// TIA Portal V20 export
// export: Created 2025-12-01T14:57:01.7824038Z, ExportSetting None, DisplayName Totally Integrated Automation Portal, DisplayVersion V20 Update 3, DisplayName TIA Portal Openness, DisplayVersion V20 Update 3, DisplayName TIA Portal Version Control Interface, DisplayVersion V20 Update 3, DisplayName STEP 7 Professional, DisplayVersion V20 Update 3, DisplayName STEP 7 Safety, DisplayVersion V20 Update 2, DisplayName WinCC Basic/Comfort/Advanced, DisplayVersion V20 Update 3, DisplayName WinCC Professional, DisplayVersion V20 Update 3, DisplayName WinCC Unified, DisplayVersion V20 Update 3
FUNCTION "FC460_TL_Merge" : Void   // FC460, LAD
{ S7_Optimized_Access := 'FALSE' }
AUTHOR : TLigero
NAME : 20160208
VERSION : 3.3
// stored: AutoNumber false, SetENOAutomatically false
   VAR_INPUT
      Mesa : UInt;
      En_Tension : Bool;
      PhsMx : Bool;
      Avance_Tx : Bool;
      Termico_Tx : Bool;
      Simul_Mx : Bool;
      AVTF_MAnt_E1 : Bool;
      AVTF_MAnt_E2 : Bool;
      PTF_Mx_MSig : Bool;
      NXT_Avance : Bool;
      V_Paro : UDInt;
      V_TOut_Tx_Mx : UDInt;
      V_CNT_pHsMx : UDInt;
      V_Salida : UDInt;
      V_Gap : UDInt;
      V_Cajas_Equ_E1 : UDInt;
      V_Cajas_Equ_E2 : UDInt;
      V_Vaciado_E1 : UDInt;
      V_Vaciado_E2 : UDInt;
   END_VAR
   VAR_OUTPUT
      PTF_Ent_M1 : Bool;
      PTF_Ent_M2 : Bool;
      AVTF_Mx_MSig : Bool;
      NXT_Descarga_Act : Bool;
   END_VAR
   VAR_IN_OUT
      Mem_CNT_Salida : Bool;
      Mem_CNT_Tmp_Paro_Tx : Bool;
      MAUX_FP_Marcha : Bool;
      MAUX_FN_PHS : Bool;
      MAUX_PRV_Carga_OK_E1 : Bool;
      MAUX_PRV_Carga_OK_E2 : Bool;
      MAUX_FP_contador_E1 : Bool;
      MAUX_FP_contador_E2 : Bool;
      MAUX_FP_En_camino_E1 : Bool;
      MAUX_FP_En_camino_E2 : Bool;
      MAUX_key_En_E1 : Bool;
      MAUX_key_En_E2 : Bool;
      MAUX_Key_por_E1_fue_usada : Bool;
      MAUX_Key_por_E2_fue_usada : Bool;
      MAUX_Caja_En_Camino_E1 : Bool;
      MAUX_Caja_En_Camino_E2 : Bool;
   END_VAR
   VAR_TEMP
      OK_Avance : Bool;
      fp_Marcha : Bool;
      fn_phs_tx : Bool;
      fp_phs_tx : Bool;
      Mem_CNT_Centrado : Bool;
      Mem_CNT_Gap : Bool;
      Error_atasco : Bool;
      TEMP_NXT_AVTF : Bool;
      TEMP_PRV_CARGA_OK : Bool;
      VaciadoE1_OK : Bool;
      VaciadoE2_OK : Bool;
      ok_tension : Bool;
   END_VAR
   VAR_TEMP   // added for the SCL form of the ladder/FBD networks
      _w1 : Bool;
   END_VAR
BEGIN

REGION Network 1: Marca General Error
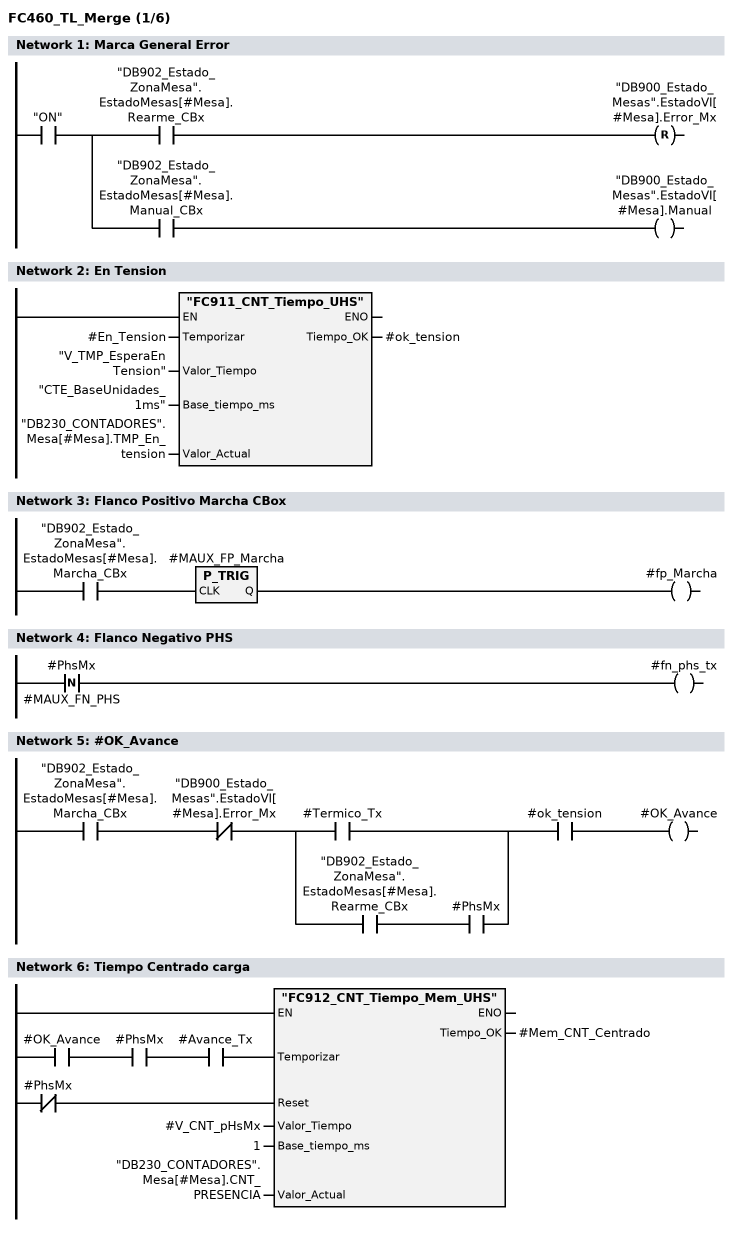
   RUNG wire#powerrail
      Contact( "ON" )
      wire#w1
      Contact( "DB902_Estado_ZonaMesa".EstadoMesas[#Mesa].Rearme_CBx )
      R_Coil( "DB900_Estado_Mesas".EstadoVI[#Mesa].Error_Mx )
   END_RUNG
   RUNG wire#w1
      Contact( "DB902_Estado_ZonaMesa".EstadoMesas[#Mesa].Manual_CBx )
      Coil( "DB900_Estado_Mesas".EstadoVI[#Mesa].Manual )
   END_RUNG
   // the same network as SCL:
   IF "ON" AND "DB902_Estado_ZonaMesa".EstadoMesas[#Mesa].Rearme_CBx THEN
       "DB900_Estado_Mesas".EstadoVI[#Mesa].Error_Mx := FALSE;
   END_IF;
   "DB900_Estado_Mesas".EstadoVI[#Mesa].Manual := "ON" AND "DB902_Estado_ZonaMesa".EstadoMesas[#Mesa].Manual_CBx;
END_REGION

REGION Network 2: En Tension
   RUNG wire#powerrail
      "FC911_CNT_Tiempo_UHS"(Temporizar := #En_Tension, Valor_Tiempo := "V_TMP_EsperaEnTension", Base_tiempo_ms := "CTE_BaseUnidades_1ms", Valor_Actual := "DB230_CONTADORES".Mesa[#Mesa].TMP_En_tension, Tiempo_OK => #ok_tension)
   END_RUNG
   // the same network as SCL:
   "FC911_CNT_Tiempo_UHS"(Temporizar := #En_Tension,
                          Valor_Tiempo := "V_TMP_EsperaEnTension",
                          Base_tiempo_ms := "CTE_BaseUnidades_1ms",
                          Valor_Actual := "DB230_CONTADORES".Mesa[#Mesa].TMP_En_tension,
                          Tiempo_OK => #ok_tension);
END_REGION

REGION Network 3: Flanco Positivo Marcha CBox
   RUNG wire#powerrail
      Contact( "DB902_Estado_ZonaMesa".EstadoMesas[#Mesa].Marcha_CBx )
      P_Trig( #MAUX_FP_Marcha )
      Coil( #fp_Marcha )
   END_RUNG
   // the same network as SCL:
   #_w1 := "DB902_Estado_ZonaMesa".EstadoMesas[#Mesa].Marcha_CBx AND NOT #MAUX_FP_Marcha;   // rising edge
   #MAUX_FP_Marcha := "DB902_Estado_ZonaMesa".EstadoMesas[#Mesa].Marcha_CBx;
   #fp_Marcha := #_w1;
END_REGION

REGION Network 4: Flanco Negativo PHS
   RUNG wire#powerrail
      N_Contact(operand := #PhsMx, bit := #MAUX_FN_PHS)
      Coil( #fn_phs_tx )
   END_RUNG
   // the same network as SCL:
   #_w1 := NOT #PhsMx AND #MAUX_FN_PHS;   // falling edge of #PhsMx
   #MAUX_FN_PHS := #PhsMx;
   #fn_phs_tx := #_w1;
END_REGION

REGION Network 5: #OK_Avance
   RUNG wire#powerrail
      Contact( "DB902_Estado_ZonaMesa".EstadoMesas[#Mesa].Marcha_CBx )
      I_Contact( "DB900_Estado_Mesas".EstadoVI[#Mesa].Error_Mx )
      wire#w1
      Contact( #Termico_Tx )
      wire#w2
      Contact( #ok_tension )
      Coil( #OK_Avance )
   END_RUNG
   RUNG wire#w1
      Contact( "DB902_Estado_ZonaMesa".EstadoMesas[#Mesa].Rearme_CBx )
      Contact( #PhsMx )
   END_RUNG wire#w2
   // the same network as SCL:
   #OK_Avance := "DB902_Estado_ZonaMesa".EstadoMesas[#Mesa].Marcha_CBx AND NOT "DB900_Estado_Mesas".EstadoVI[#Mesa].Error_Mx AND (#Termico_Tx OR ("DB902_Estado_ZonaMesa".EstadoMesas[#Mesa].Rearme_CBx AND #PhsMx)) AND #ok_tension;
END_REGION

REGION Network 6: Tiempo Centrado carga
   RUNG wire#powerrail
      "FC912_CNT_Tiempo_Mem_UHS"(Temporizar := wire#w1, Reset := wire#w2, Valor_Tiempo := #V_CNT_pHsMx, Base_tiempo_ms := 1, Valor_Actual := "DB230_CONTADORES".Mesa[#Mesa].CNT_PRESENCIA, Tiempo_OK => #Mem_CNT_Centrado)
   END_RUNG
   RUNG wire#powerrail
      Contact( #OK_Avance )
      Contact( #PhsMx )
      Contact( #Avance_Tx )
   END_RUNG wire#w1
   RUNG wire#powerrail
      I_Contact( #PhsMx )
   END_RUNG wire#w2
   // the same network as SCL:
   "FC912_CNT_Tiempo_Mem_UHS"(Temporizar := #OK_Avance AND #PhsMx AND #Avance_Tx,
                           Reset := NOT #PhsMx,
                           Valor_Tiempo := #V_CNT_pHsMx,
                           Base_tiempo_ms := 1,
                           Valor_Actual := "DB230_CONTADORES".Mesa[#Mesa].CNT_PRESENCIA,
                           Tiempo_OK => #Mem_CNT_Centrado);
END_REGION

REGION Network 7: Tiempo Centrado carga
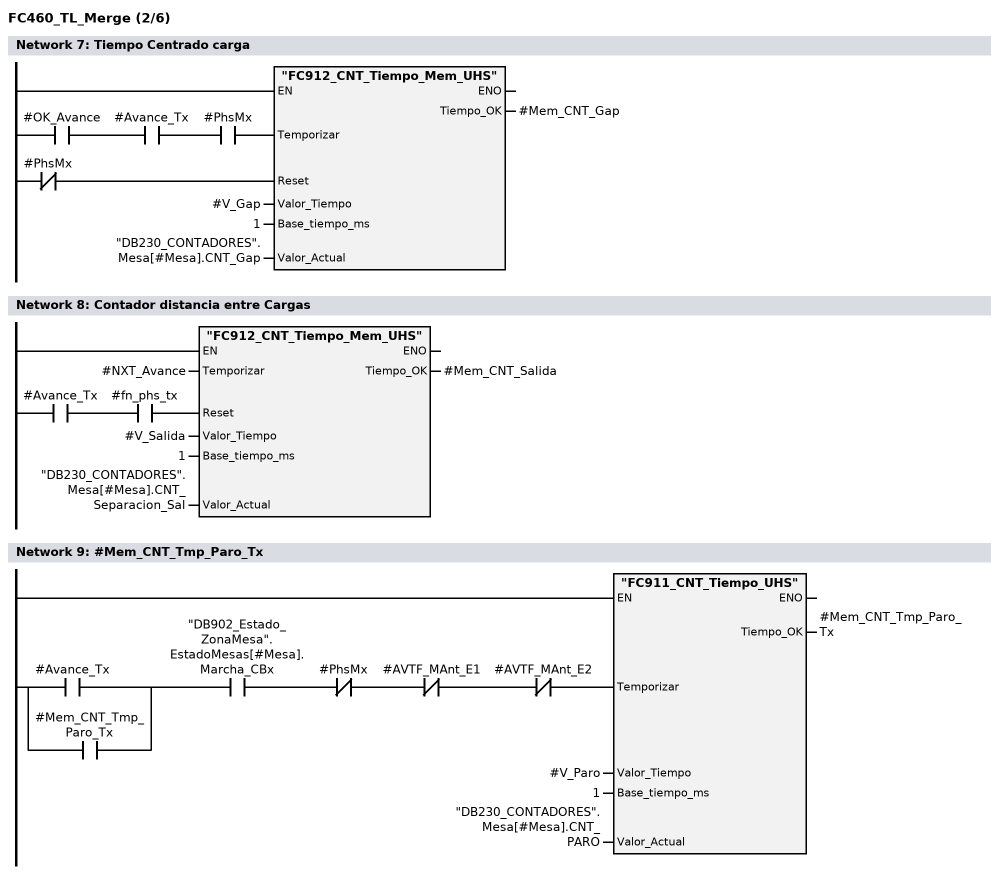
   RUNG wire#powerrail
      "FC912_CNT_Tiempo_Mem_UHS"(Temporizar := wire#w1, Reset := wire#w2, Valor_Tiempo := #V_Gap, Base_tiempo_ms := 1, Valor_Actual := "DB230_CONTADORES".Mesa[#Mesa].CNT_Gap, Tiempo_OK => #Mem_CNT_Gap)
   END_RUNG
   RUNG wire#powerrail
      Contact( #OK_Avance )
      Contact( #Avance_Tx )
      Contact( #PhsMx )
   END_RUNG wire#w1
   RUNG wire#powerrail
      I_Contact( #PhsMx )
   END_RUNG wire#w2
   // the same network as SCL:
   "FC912_CNT_Tiempo_Mem_UHS"(Temporizar := #OK_Avance AND #Avance_Tx AND #PhsMx,
                           Reset := NOT #PhsMx,
                           Valor_Tiempo := #V_Gap,
                           Base_tiempo_ms := 1,
                           Valor_Actual := "DB230_CONTADORES".Mesa[#Mesa].CNT_Gap,
                           Tiempo_OK => #Mem_CNT_Gap);
END_REGION

REGION Network 8: Contador distancia entre Cargas
   RUNG wire#powerrail
      "FC912_CNT_Tiempo_Mem_UHS"(Reset := wire#w1, Temporizar := #NXT_Avance, Valor_Tiempo := #V_Salida, Base_tiempo_ms := 1, Valor_Actual := "DB230_CONTADORES".Mesa[#Mesa].CNT_Separacion_Sal, Tiempo_OK => #Mem_CNT_Salida)
   END_RUNG
   RUNG wire#powerrail
      Contact( #Avance_Tx )
      Contact( #fn_phs_tx )
   END_RUNG wire#w1
   // the same network as SCL:
   "FC912_CNT_Tiempo_Mem_UHS"(Temporizar := #NXT_Avance,
                           Reset := #Avance_Tx AND #fn_phs_tx,
                           Valor_Tiempo := #V_Salida,
                           Base_tiempo_ms := 1,
                           Valor_Actual := "DB230_CONTADORES".Mesa[#Mesa].CNT_Separacion_Sal,
                           Tiempo_OK => #Mem_CNT_Salida);
END_REGION

REGION Network 9: #Mem_CNT_Tmp_Paro_Tx
   RUNG wire#powerrail
      "FC911_CNT_Tiempo_UHS"(Temporizar := wire#w2, Valor_Tiempo := #V_Paro, Base_tiempo_ms := 1, Valor_Actual := "DB230_CONTADORES".Mesa[#Mesa].CNT_PARO, Tiempo_OK => #Mem_CNT_Tmp_Paro_Tx)
   END_RUNG
   RUNG wire#powerrail
      Contact( #Avance_Tx )
      wire#w1
      Contact( "DB902_Estado_ZonaMesa".EstadoMesas[#Mesa].Marcha_CBx )
      I_Contact( #PhsMx )
      I_Contact( #AVTF_MAnt_E1 )
      I_Contact( #AVTF_MAnt_E2 )
   END_RUNG wire#w2
   RUNG wire#powerrail
      Contact( #Mem_CNT_Tmp_Paro_Tx )
   END_RUNG wire#w1
   // the same network as SCL:
   "FC911_CNT_Tiempo_UHS"(Temporizar := (#Avance_Tx OR #Mem_CNT_Tmp_Paro_Tx) AND "DB902_Estado_ZonaMesa".EstadoMesas[#Mesa].Marcha_CBx AND NOT #PhsMx AND NOT #AVTF_MAnt_E1 AND NOT #AVTF_MAnt_E2,
                          Valor_Tiempo := #V_Paro,
                          Base_tiempo_ms := 1,
                          Valor_Actual := "DB230_CONTADORES".Mesa[#Mesa].CNT_PARO,
                          Tiempo_OK => #Mem_CNT_Tmp_Paro_Tx);
END_REGION

REGION Network 10: #MA_AV_13_T_MX
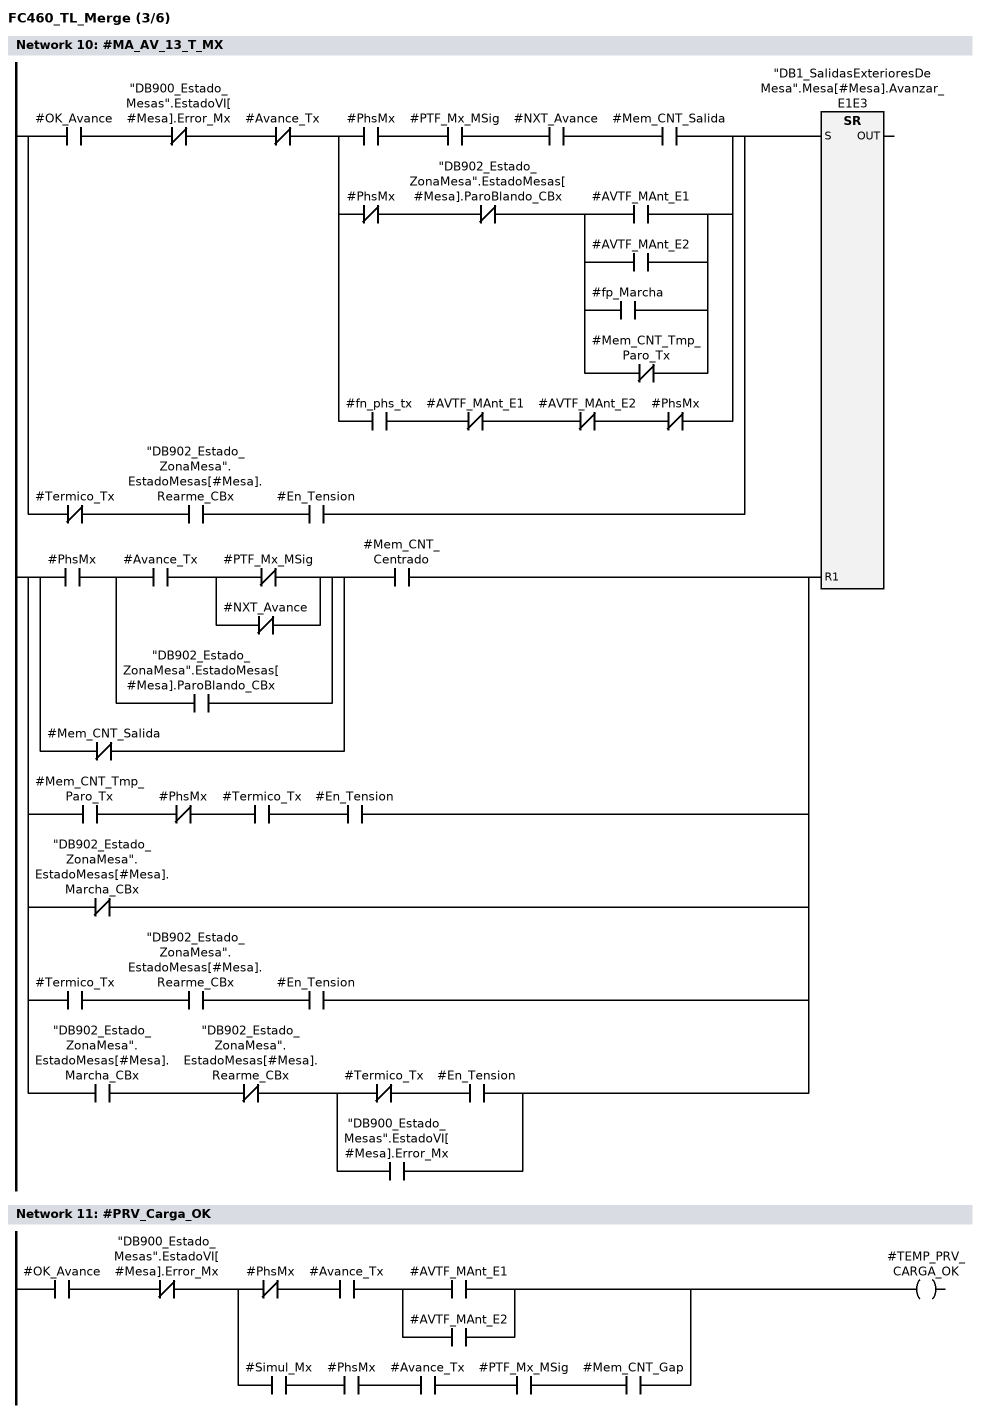
   RUNG wire#powerrail
      Contact( #OK_Avance )
      I_Contact( "DB900_Estado_Mesas".EstadoVI[#Mesa].Error_Mx )
      I_Contact( #Avance_Tx )
      wire#w1
      Contact( #PhsMx )
      Contact( #PTF_Mx_MSig )
      Contact( #NXT_Avance )
      Contact( #Mem_CNT_Salida )
      wire#w2
      S_SR(operand := "DB1_SalidasExterioresDeMesa".Mesa[#Mesa].Avanzar_E1E3, r1 := wire#w8)
   END_RUNG
   RUNG wire#w1
      I_Contact( #PhsMx )
      I_Contact( "DB902_Estado_ZonaMesa".EstadoMesas[#Mesa].ParoBlando_CBx )
      wire#w3
      Contact( #AVTF_MAnt_E1 )
   END_RUNG wire#w2
   RUNG wire#w3
      Contact( #AVTF_MAnt_E2 )
   END_RUNG wire#w2
   RUNG wire#w3
      Contact( #fp_Marcha )
   END_RUNG wire#w2
   RUNG wire#w3
      I_Contact( #Mem_CNT_Tmp_Paro_Tx )
   END_RUNG wire#w2
   RUNG wire#w1
      Contact( #fn_phs_tx )
      I_Contact( #AVTF_MAnt_E1 )
      I_Contact( #AVTF_MAnt_E2 )
      I_Contact( #PhsMx )
   END_RUNG wire#w2
   RUNG wire#powerrail
      I_Contact( #Termico_Tx )
      Contact( "DB902_Estado_ZonaMesa".EstadoMesas[#Mesa].Rearme_CBx )
      Contact( #En_Tension )
   END_RUNG wire#w2
   RUNG wire#powerrail
      Contact( #PhsMx )
      wire#w4
      Contact( #Avance_Tx )
      wire#w5
      I_Contact( #PTF_Mx_MSig )
      wire#w6
      Contact( #Mem_CNT_Centrado )
   END_RUNG wire#w8
   RUNG wire#w5
      I_Contact( #NXT_Avance )
   END_RUNG wire#w6
   RUNG wire#w4
      Contact( "DB902_Estado_ZonaMesa".EstadoMesas[#Mesa].ParoBlando_CBx )
   END_RUNG wire#w6
   RUNG wire#powerrail
      I_Contact( #Mem_CNT_Salida )
   END_RUNG wire#w6
   RUNG wire#powerrail
      Contact( #Mem_CNT_Tmp_Paro_Tx )
      I_Contact( #PhsMx )
      Contact( #Termico_Tx )
      Contact( #En_Tension )
   END_RUNG wire#w8
   RUNG wire#powerrail
      I_Contact( "DB902_Estado_ZonaMesa".EstadoMesas[#Mesa].Marcha_CBx )
   END_RUNG wire#w8
   RUNG wire#powerrail
      Contact( #Termico_Tx )
      Contact( "DB902_Estado_ZonaMesa".EstadoMesas[#Mesa].Rearme_CBx )
      Contact( #En_Tension )
   END_RUNG wire#w8
   RUNG wire#powerrail
      Contact( "DB902_Estado_ZonaMesa".EstadoMesas[#Mesa].Marcha_CBx )
      I_Contact( "DB902_Estado_ZonaMesa".EstadoMesas[#Mesa].Rearme_CBx )
      wire#w7
      I_Contact( #Termico_Tx )
      Contact( #En_Tension )
   END_RUNG wire#w8
   RUNG wire#w7
      Contact( "DB900_Estado_Mesas".EstadoVI[#Mesa].Error_Mx )
   END_RUNG wire#w8
   // the same network as SCL:
   #_w1 := (((#PhsMx AND ((#Avance_Tx AND (NOT #PTF_Mx_MSig OR NOT #NXT_Avance)) OR "DB902_Estado_ZonaMesa".EstadoMesas[#Mesa].ParoBlando_CBx)) OR NOT #Mem_CNT_Salida) AND #Mem_CNT_Centrado) OR (#Mem_CNT_Tmp_Paro_Tx AND NOT #PhsMx AND #Termico_Tx AND #En_Tension) OR NOT "DB902_Estado_ZonaMesa".EstadoMesas[#Mesa].Marcha_CBx OR (#Termico_Tx AND "DB902_Estado_ZonaMesa".EstadoMesas[#Mesa].Rearme_CBx AND #En_Tension) OR ("DB902_Estado_ZonaMesa".EstadoMesas[#Mesa].Marcha_CBx AND NOT "DB902_Estado_ZonaMesa".EstadoMesas[#Mesa].Rearme_CBx AND ((NOT #Termico_Tx AND #En_Tension) OR "DB900_Estado_Mesas".EstadoVI[#Mesa].Error_Mx));
   IF (#OK_Avance AND NOT "DB900_Estado_Mesas".EstadoVI[#Mesa].Error_Mx AND NOT #Avance_Tx AND ((#PhsMx AND #PTF_Mx_MSig AND #NXT_Avance AND #Mem_CNT_Salida) OR (NOT #PhsMx AND NOT "DB902_Estado_ZonaMesa".EstadoMesas[#Mesa].ParoBlando_CBx AND (#AVTF_MAnt_E1 OR #AVTF_MAnt_E2 OR #fp_Marcha OR NOT #Mem_CNT_Tmp_Paro_Tx)) OR (#fn_phs_tx AND NOT #AVTF_MAnt_E1 AND NOT #AVTF_MAnt_E2 AND NOT #PhsMx))) OR (NOT #Termico_Tx AND "DB902_Estado_ZonaMesa".EstadoMesas[#Mesa].Rearme_CBx AND #En_Tension) THEN
       "DB1_SalidasExterioresDeMesa".Mesa[#Mesa].Avanzar_E1E3 := TRUE;   // SR flip-flop
   END_IF;
   IF #_w1 THEN "DB1_SalidasExterioresDeMesa".Mesa[#Mesa].Avanzar_E1E3 := FALSE; END_IF;
END_REGION

REGION Network 11: #PRV_Carga_OK
   RUNG wire#powerrail
      Contact( #OK_Avance )
      I_Contact( "DB900_Estado_Mesas".EstadoVI[#Mesa].Error_Mx )
      wire#w1
      I_Contact( #PhsMx )
      Contact( #Avance_Tx )
      wire#w2
      Contact( #AVTF_MAnt_E1 )
      wire#w3
      Coil( #TEMP_PRV_CARGA_OK )
   END_RUNG
   RUNG wire#w2
      Contact( #AVTF_MAnt_E2 )
   END_RUNG wire#w3
   RUNG wire#w1
      Contact( #Simul_Mx )
      Contact( #PhsMx )
      Contact( #Avance_Tx )
      Contact( #PTF_Mx_MSig )
      Contact( #Mem_CNT_Gap )
   END_RUNG wire#w3
   // the same network as SCL:
   #TEMP_PRV_CARGA_OK := #OK_Avance AND NOT "DB900_Estado_Mesas".EstadoVI[#Mesa].Error_Mx AND ((NOT #PhsMx AND #Avance_Tx AND (#AVTF_MAnt_E1 OR #AVTF_MAnt_E2)) OR (#Simul_Mx AND #PhsMx AND #Avance_Tx AND #PTF_Mx_MSig AND #Mem_CNT_Gap));
END_REGION

REGION Network 12: #NXT_AVTF
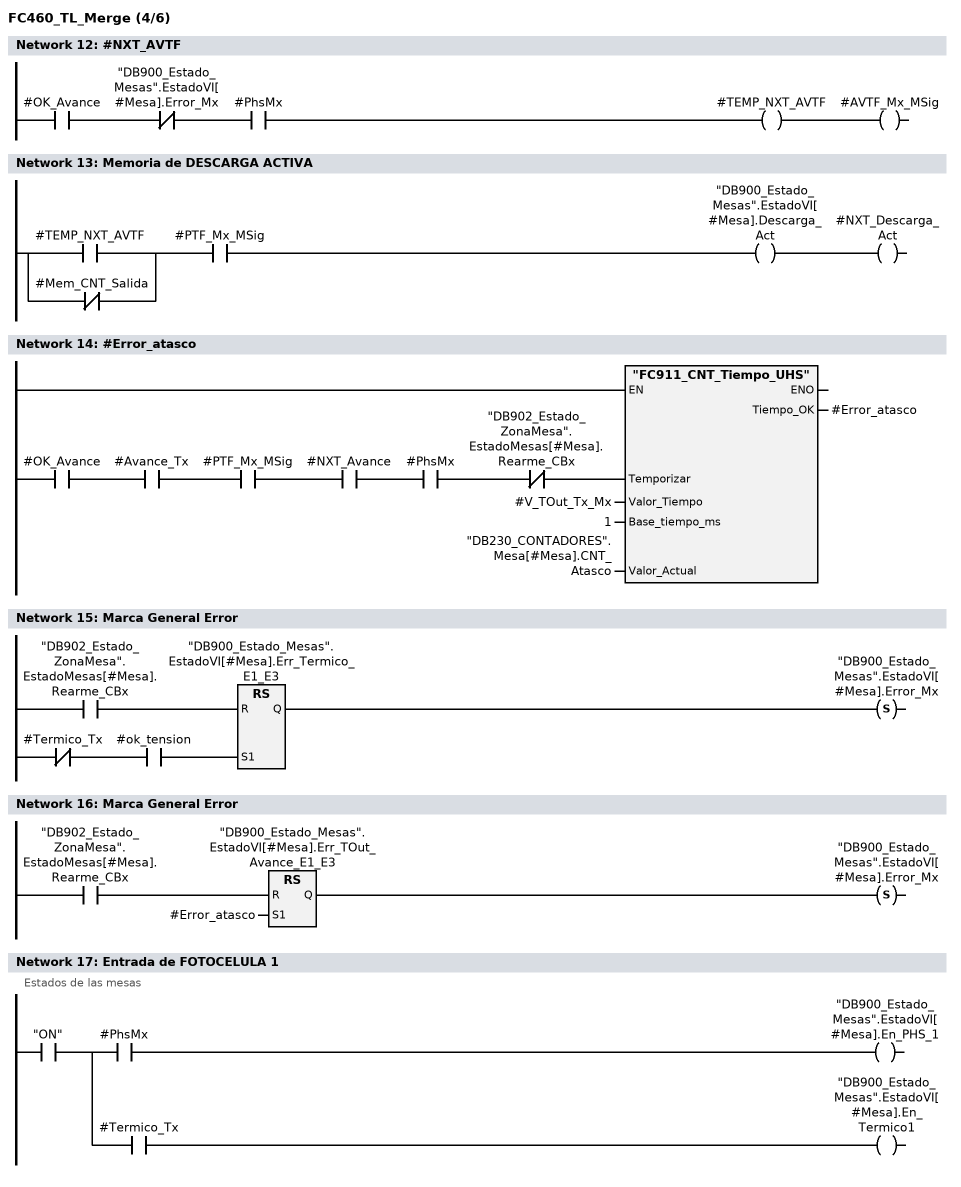
   RUNG wire#powerrail
      Contact( #OK_Avance )
      I_Contact( "DB900_Estado_Mesas".EstadoVI[#Mesa].Error_Mx )
      Contact( #PhsMx )
      Coil( #TEMP_NXT_AVTF )
      Coil( #AVTF_Mx_MSig )
   END_RUNG
   // the same network as SCL:
   #TEMP_NXT_AVTF := #OK_Avance AND NOT "DB900_Estado_Mesas".EstadoVI[#Mesa].Error_Mx AND #PhsMx;
   #AVTF_Mx_MSig := #TEMP_NXT_AVTF;
END_REGION

REGION Network 13: Memoria de DESCARGA ACTIVA
   RUNG wire#powerrail
      Contact( #TEMP_NXT_AVTF )
      wire#w1
      Contact( #PTF_Mx_MSig )
      Coil( "DB900_Estado_Mesas".EstadoVI[#Mesa].Descarga_Act )
      Coil( #NXT_Descarga_Act )
   END_RUNG
   RUNG wire#powerrail
      I_Contact( #Mem_CNT_Salida )
   END_RUNG wire#w1
   // the same network as SCL:
   "DB900_Estado_Mesas".EstadoVI[#Mesa].Descarga_Act := (#TEMP_NXT_AVTF OR NOT #Mem_CNT_Salida) AND #PTF_Mx_MSig;
   #NXT_Descarga_Act := (#TEMP_NXT_AVTF OR NOT #Mem_CNT_Salida) AND #PTF_Mx_MSig;
END_REGION

REGION Network 14: #Error_atasco
   RUNG wire#powerrail
      "FC911_CNT_Tiempo_UHS"(Temporizar := wire#w1, Valor_Tiempo := #V_TOut_Tx_Mx, Base_tiempo_ms := 1, Valor_Actual := "DB230_CONTADORES".Mesa[#Mesa].CNT_Atasco, Tiempo_OK => #Error_atasco)
   END_RUNG
   RUNG wire#powerrail
      Contact( #OK_Avance )
      Contact( #Avance_Tx )
      Contact( #PTF_Mx_MSig )
      Contact( #NXT_Avance )
      Contact( #PhsMx )
      I_Contact( "DB902_Estado_ZonaMesa".EstadoMesas[#Mesa].Rearme_CBx )
   END_RUNG wire#w1
   // the same network as SCL:
   "FC911_CNT_Tiempo_UHS"(Temporizar := #OK_Avance AND #Avance_Tx AND #PTF_Mx_MSig AND #NXT_Avance AND #PhsMx AND NOT "DB902_Estado_ZonaMesa".EstadoMesas[#Mesa].Rearme_CBx,
                          Valor_Tiempo := #V_TOut_Tx_Mx,
                          Base_tiempo_ms := 1,
                          Valor_Actual := "DB230_CONTADORES".Mesa[#Mesa].CNT_Atasco,
                          Tiempo_OK => #Error_atasco);
END_REGION

REGION Network 15: Marca General Error
   RUNG wire#powerrail
      Contact( "DB902_Estado_ZonaMesa".EstadoMesas[#Mesa].Rearme_CBx )
      S_RS(operand := "DB900_Estado_Mesas".EstadoVI[#Mesa].Err_Termico_E1_E3, s1 := wire#w1)
      S_Coil( "DB900_Estado_Mesas".EstadoVI[#Mesa].Error_Mx )
   END_RUNG
   RUNG wire#powerrail
      I_Contact( #Termico_Tx )
      Contact( #ok_tension )
   END_RUNG wire#w1
   // the same network as SCL:
   IF "DB902_Estado_ZonaMesa".EstadoMesas[#Mesa].Rearme_CBx THEN
       "DB900_Estado_Mesas".EstadoVI[#Mesa].Err_Termico_E1_E3 := FALSE;   // RS flip-flop
   END_IF;
   IF NOT #Termico_Tx AND #ok_tension THEN
       "DB900_Estado_Mesas".EstadoVI[#Mesa].Err_Termico_E1_E3 := TRUE;
   END_IF;
   IF "DB900_Estado_Mesas".EstadoVI[#Mesa].Err_Termico_E1_E3 THEN
       "DB900_Estado_Mesas".EstadoVI[#Mesa].Error_Mx := TRUE;
   END_IF;
END_REGION

REGION Network 16: Marca General Error
   RUNG wire#powerrail
      Contact( "DB902_Estado_ZonaMesa".EstadoMesas[#Mesa].Rearme_CBx )
      S_RS(operand := "DB900_Estado_Mesas".EstadoVI[#Mesa].Err_TOut_Avance_E1_E3, s1 := #Error_atasco)
      S_Coil( "DB900_Estado_Mesas".EstadoVI[#Mesa].Error_Mx )
   END_RUNG
   // the same network as SCL:
   IF "DB902_Estado_ZonaMesa".EstadoMesas[#Mesa].Rearme_CBx THEN
       "DB900_Estado_Mesas".EstadoVI[#Mesa].Err_TOut_Avance_E1_E3 := FALSE;   // RS flip-flop
   END_IF;
   IF #Error_atasco THEN "DB900_Estado_Mesas".EstadoVI[#Mesa].Err_TOut_Avance_E1_E3 := TRUE; END_IF;
   IF "DB900_Estado_Mesas".EstadoVI[#Mesa].Err_TOut_Avance_E1_E3 THEN
       "DB900_Estado_Mesas".EstadoVI[#Mesa].Error_Mx := TRUE;
   END_IF;
END_REGION

REGION Network 17: Entrada de FOTOCELULA 1
   // Estados de las mesas
   RUNG wire#powerrail
      Contact( "ON" )
      wire#w1
      Contact( #PhsMx )
      Coil( "DB900_Estado_Mesas".EstadoVI[#Mesa].En_PHS_1 )
   END_RUNG
   RUNG wire#w1
      Contact( #Termico_Tx )
      Coil( "DB900_Estado_Mesas".EstadoVI[#Mesa].En_Termico1 )
   END_RUNG
   // the same network as SCL:
   "DB900_Estado_Mesas".EstadoVI[#Mesa].En_PHS_1 := "ON" AND #PhsMx;
   "DB900_Estado_Mesas".EstadoVI[#Mesa].En_Termico1 := "ON" AND #Termico_Tx;
END_REGION

REGION Network 18: ESTADOS MESA 1
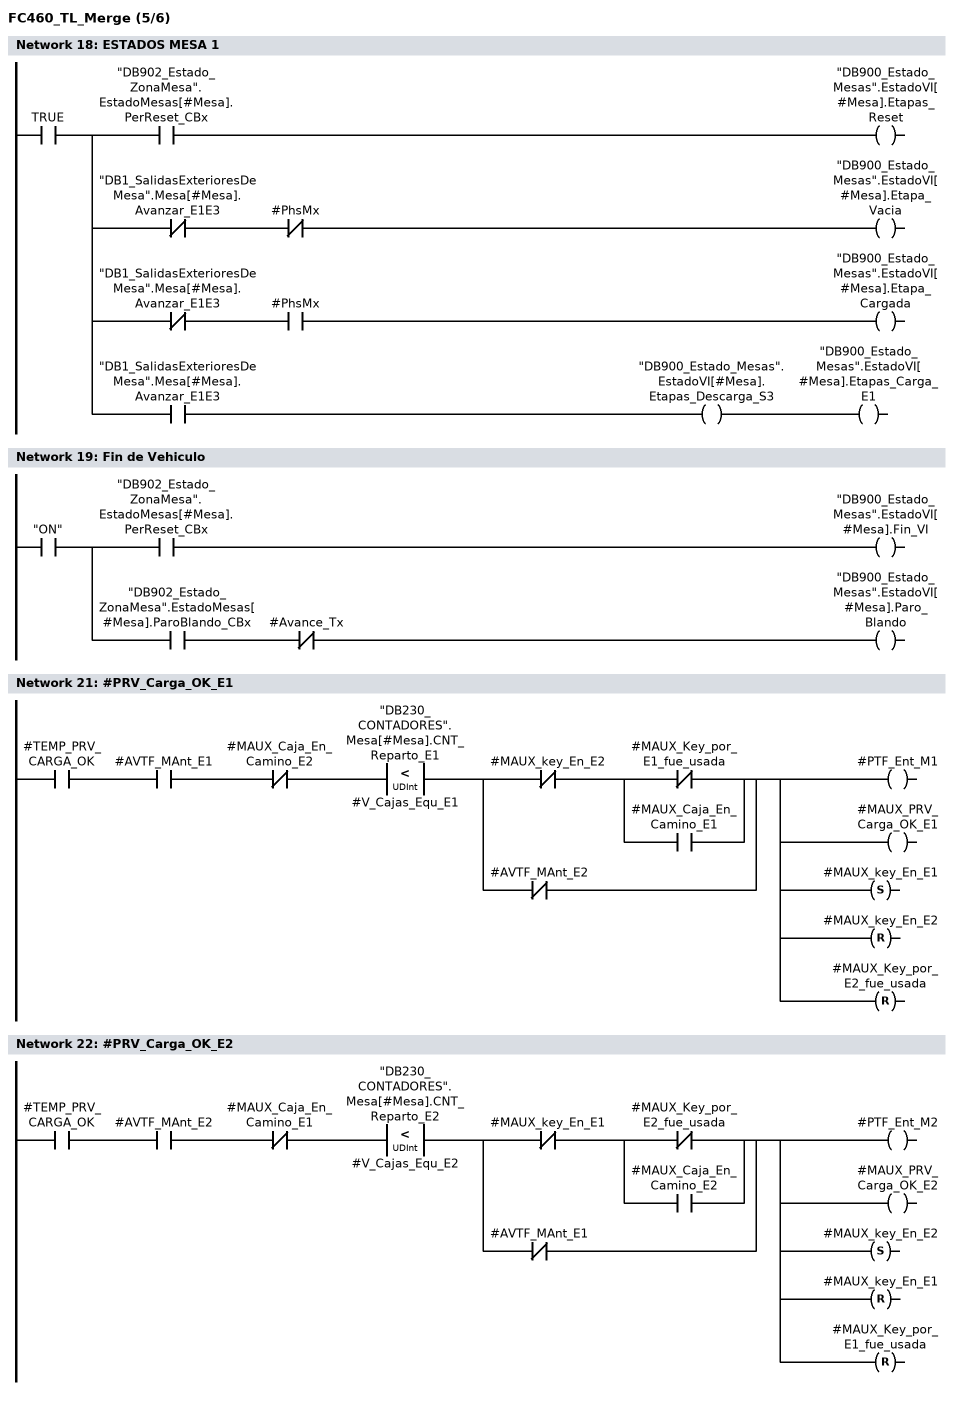
   RUNG wire#powerrail
      Contact( TRUE )
      wire#w1
      Contact( "DB902_Estado_ZonaMesa".EstadoMesas[#Mesa].PerReset_CBx )
      Coil( "DB900_Estado_Mesas".EstadoVI[#Mesa].Etapas_Reset )
   END_RUNG
   RUNG wire#w1
      I_Contact( "DB1_SalidasExterioresDeMesa".Mesa[#Mesa].Avanzar_E1E3 )
      I_Contact( #PhsMx )
      Coil( "DB900_Estado_Mesas".EstadoVI[#Mesa].Etapa_Vacia )
   END_RUNG
   RUNG wire#w1
      I_Contact( "DB1_SalidasExterioresDeMesa".Mesa[#Mesa].Avanzar_E1E3 )
      Contact( #PhsMx )
      Coil( "DB900_Estado_Mesas".EstadoVI[#Mesa].Etapa_Cargada )
   END_RUNG
   RUNG wire#w1
      Contact( "DB1_SalidasExterioresDeMesa".Mesa[#Mesa].Avanzar_E1E3 )
      Coil( "DB900_Estado_Mesas".EstadoVI[#Mesa].Etapas_Descarga_S3 )
      Coil( "DB900_Estado_Mesas".EstadoVI[#Mesa].Etapas_Carga_E1 )
   END_RUNG
   // the same network as SCL:
   "DB900_Estado_Mesas".EstadoVI[#Mesa].Etapas_Reset := TRUE AND "DB902_Estado_ZonaMesa".EstadoMesas[#Mesa].PerReset_CBx;
   "DB900_Estado_Mesas".EstadoVI[#Mesa].Etapa_Vacia := TRUE AND NOT "DB1_SalidasExterioresDeMesa".Mesa[#Mesa].Avanzar_E1E3 AND NOT #PhsMx;
   "DB900_Estado_Mesas".EstadoVI[#Mesa].Etapa_Cargada := TRUE AND NOT "DB1_SalidasExterioresDeMesa".Mesa[#Mesa].Avanzar_E1E3 AND #PhsMx;
   #_w1 := TRUE AND "DB1_SalidasExterioresDeMesa".Mesa[#Mesa].Avanzar_E1E3;
   "DB900_Estado_Mesas".EstadoVI[#Mesa].Etapas_Descarga_S3 := #_w1;
   "DB900_Estado_Mesas".EstadoVI[#Mesa].Etapas_Carga_E1 := #_w1;
END_REGION

REGION Network 19: Fin de Vehiculo
   RUNG wire#powerrail
      Contact( "ON" )
      wire#w1
      Contact( "DB902_Estado_ZonaMesa".EstadoMesas[#Mesa].PerReset_CBx )
      Coil( "DB900_Estado_Mesas".EstadoVI[#Mesa].Fin_VI )
   END_RUNG
   RUNG wire#w1
      Contact( "DB902_Estado_ZonaMesa".EstadoMesas[#Mesa].ParoBlando_CBx )
      I_Contact( #Avance_Tx )
      Coil( "DB900_Estado_Mesas".EstadoVI[#Mesa].Paro_Blando )
   END_RUNG
   // the same network as SCL:
   "DB900_Estado_Mesas".EstadoVI[#Mesa].Fin_VI := "ON" AND "DB902_Estado_ZonaMesa".EstadoMesas[#Mesa].PerReset_CBx;
   "DB900_Estado_Mesas".EstadoVI[#Mesa].Paro_Blando := "ON" AND "DB902_Estado_ZonaMesa".EstadoMesas[#Mesa].ParoBlando_CBx AND NOT #Avance_Tx;
END_REGION

REGION Network 20: Gestion de cruce
END_REGION

REGION Network 21: #PRV_Carga_OK_E1
   RUNG wire#powerrail
      Contact( #TEMP_PRV_CARGA_OK )
      Contact( #AVTF_MAnt_E1 )
      I_Contact( #MAUX_Caja_En_Camino_E2 )
      { S7_Templates := "SrcType := UDInt" } LT_Contact(in1 := "DB230_CONTADORES".Mesa[#Mesa].CNT_Reparto_E1, in2 := #V_Cajas_Equ_E1)
      wire#w1
      I_Contact( #MAUX_key_En_E2 )
      wire#w2
      I_Contact( #MAUX_Key_por_E1_fue_usada )
      wire#w3
      Coil( #PTF_Ent_M1 )
   END_RUNG
   RUNG wire#w2
      Contact( #MAUX_Caja_En_Camino_E1 )
   END_RUNG wire#w3
   RUNG wire#w1
      I_Contact( #AVTF_MAnt_E2 )
   END_RUNG wire#w3
   RUNG wire#w3
      Coil( #MAUX_PRV_Carga_OK_E1 )
   END_RUNG
   RUNG wire#w3
      S_Coil( #MAUX_key_En_E1 )
   END_RUNG
   RUNG wire#w3
      R_Coil( #MAUX_key_En_E2 )
   END_RUNG
   RUNG wire#w3
      R_Coil( #MAUX_Key_por_E2_fue_usada )
   END_RUNG
   // the same network as SCL:
   #PTF_Ent_M1 := #TEMP_PRV_CARGA_OK AND #AVTF_MAnt_E1 AND NOT #MAUX_Caja_En_Camino_E2 AND ("DB230_CONTADORES".Mesa[#Mesa].CNT_Reparto_E1 < #V_Cajas_Equ_E1) AND ((NOT #MAUX_key_En_E2 AND (NOT #MAUX_Key_por_E1_fue_usada OR #MAUX_Caja_En_Camino_E1)) OR NOT #AVTF_MAnt_E2);
   #MAUX_PRV_Carga_OK_E1 := #PTF_Ent_M1;
   IF #PTF_Ent_M1 THEN
       #MAUX_key_En_E1 := TRUE;
       #MAUX_key_En_E2 := FALSE;
       #MAUX_Key_por_E2_fue_usada := FALSE;
   END_IF;
END_REGION

REGION Network 22: #PRV_Carga_OK_E2
   RUNG wire#powerrail
      Contact( #TEMP_PRV_CARGA_OK )
      Contact( #AVTF_MAnt_E2 )
      I_Contact( #MAUX_Caja_En_Camino_E1 )
      { S7_Templates := "SrcType := UDInt" } LT_Contact(in1 := "DB230_CONTADORES".Mesa[#Mesa].CNT_Reparto_E2, in2 := #V_Cajas_Equ_E2)
      wire#w1
      I_Contact( #MAUX_key_En_E1 )
      wire#w2
      I_Contact( #MAUX_Key_por_E2_fue_usada )
      wire#w3
      Coil( #PTF_Ent_M2 )
   END_RUNG
   RUNG wire#w2
      Contact( #MAUX_Caja_En_Camino_E2 )
   END_RUNG wire#w3
   RUNG wire#w1
      I_Contact( #AVTF_MAnt_E1 )
   END_RUNG wire#w3
   RUNG wire#w3
      Coil( #MAUX_PRV_Carga_OK_E2 )
   END_RUNG
   RUNG wire#w3
      S_Coil( #MAUX_key_En_E2 )
   END_RUNG
   RUNG wire#w3
      R_Coil( #MAUX_key_En_E1 )
   END_RUNG
   RUNG wire#w3
      R_Coil( #MAUX_Key_por_E1_fue_usada )
   END_RUNG
   // the same network as SCL:
   #PTF_Ent_M2 := #TEMP_PRV_CARGA_OK AND #AVTF_MAnt_E2 AND NOT #MAUX_Caja_En_Camino_E1 AND ("DB230_CONTADORES".Mesa[#Mesa].CNT_Reparto_E2 < #V_Cajas_Equ_E2) AND ((NOT #MAUX_key_En_E1 AND (NOT #MAUX_Key_por_E2_fue_usada OR #MAUX_Caja_En_Camino_E2)) OR NOT #AVTF_MAnt_E1);
   #MAUX_PRV_Carga_OK_E2 := #PTF_Ent_M2;
   IF #PTF_Ent_M2 THEN
       #MAUX_key_En_E2 := TRUE;
       #MAUX_key_En_E1 := FALSE;
       #MAUX_Key_por_E1_fue_usada := FALSE;
   END_IF;
END_REGION

NETWORK
TITLE = Contador de cajas permitidas por E1
      A     #MAUX_PRV_Carga_OK_E1;
      FN    #MAUX_FP_contador_E1;
      JCN   cont1;

      L     "DB230_CONTADORES".Mesa[#Mesa].CNT_Reparto_E1;
      L     1;
      +I;
      T     "DB230_CONTADORES".Mesa[#Mesa].CNT_Reparto_E1;
//si no hay aviso de transferencia por E2, entonces se deja entrar otra vez por E1. Aunque ya se haya cumplido el
//contador. y si eso sucede, se tiene que resetear el key usada, de lo contrario, no dejariamos entrar de nnuevo
      R     #MAUX_Key_por_E1_fue_usada;

cont1:NOP   0;

      A     #MAUX_PRV_Carga_OK_E2;
      FN    #MAUX_FP_contador_E2;
      JCN   cont2;

      L     "DB230_CONTADORES".Mesa[#Mesa].CNT_Reparto_E2;
      L     1;
      +I;
      T     "DB230_CONTADORES".Mesa[#Mesa].CNT_Reparto_E2;
//si no hay aviso de transferencia por E2, entonces se deja entrar otra vez por E1. Aunque ya se haya cumplido el
//contador. y si eso sucede, se tiene que resetear el key usada, de lo contrario, no dejariamos entrar de nnuevo
      R     #MAUX_Key_por_E2_fue_usada;



cont2:NOP   0;

//llegando al maximo tenemos que resetear el valor
      L     "DB230_CONTADORES".Mesa[#Mesa].CNT_Reparto_E1;
      L     #V_Cajas_Equ_E1;
      >=I;
      JCN   borr1;
      L     0;
      T     "DB230_CONTADORES".Mesa[#Mesa].CNT_Reparto_E1;

      R     #MAUX_key_En_E1;
      S     #MAUX_Key_por_E1_fue_usada;
borr1:NOP   0;

//llegando al maximo tenemos que resetear el valor
      L     "DB230_CONTADORES".Mesa[#Mesa].CNT_Reparto_E2;
      L     #V_Cajas_Equ_E2;
      >=I;
      JCN   borr2;
      L     0;
      T     "DB230_CONTADORES".Mesa[#Mesa].CNT_Reparto_E2;

      R     #MAUX_key_En_E2;
      S     #MAUX_Key_por_E2_fue_usada;
borr2:NOP   0;





REGION Network 24: Caja en caminno por E1. Nada puede entrar por E2
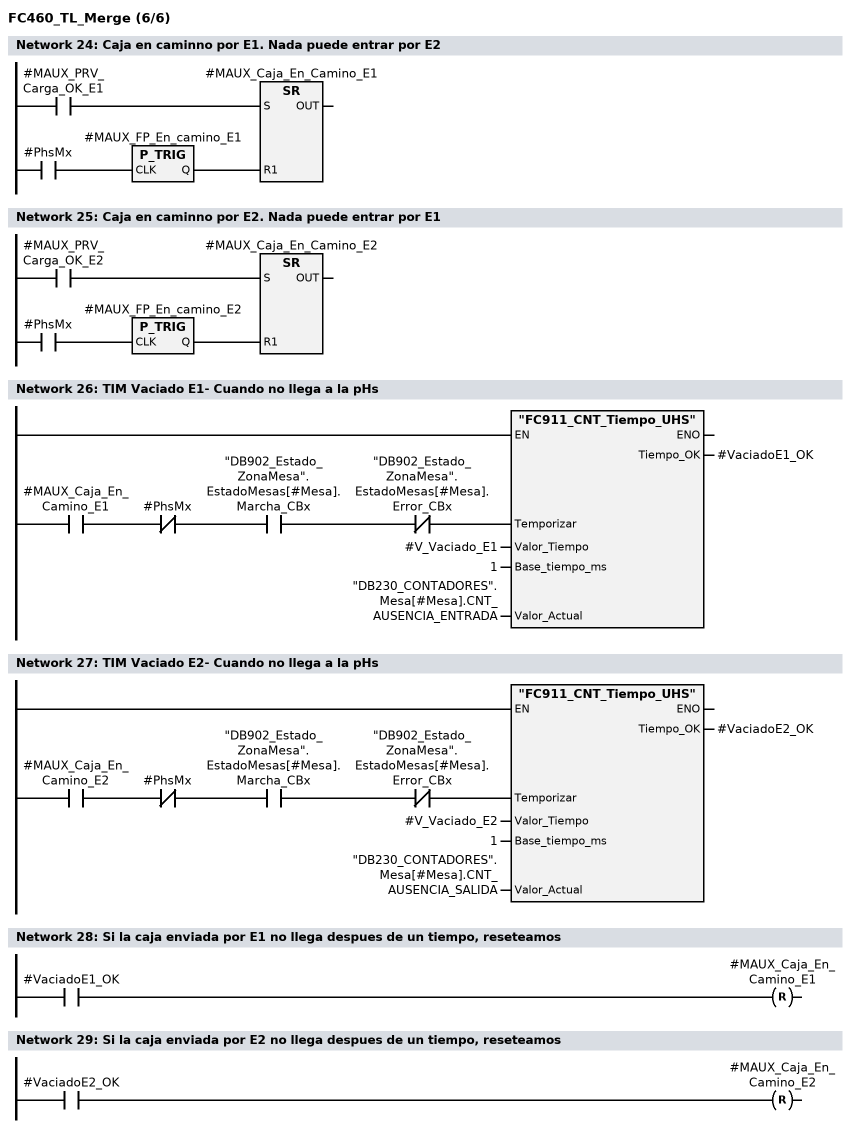
   RUNG wire#powerrail
      Contact( #MAUX_PRV_Carga_OK_E1 )
      S_SR(operand := #MAUX_Caja_En_Camino_E1, r1 := wire#w1)
   END_RUNG
   RUNG wire#powerrail
      Contact( #PhsMx )
      P_Trig( #MAUX_FP_En_camino_E1 )
   END_RUNG wire#w1
   // the same network as SCL:
   #_w1 := #PhsMx AND NOT #MAUX_FP_En_camino_E1;   // rising edge
   #MAUX_FP_En_camino_E1 := #PhsMx;
   IF #MAUX_PRV_Carga_OK_E1 THEN
       #MAUX_Caja_En_Camino_E1 := TRUE;   // SR flip-flop
   END_IF;
   IF #_w1 THEN #MAUX_Caja_En_Camino_E1 := FALSE; END_IF;
END_REGION

REGION Network 25: Caja en caminno por E2. Nada puede entrar por E1
   RUNG wire#powerrail
      Contact( #MAUX_PRV_Carga_OK_E2 )
      S_SR(operand := #MAUX_Caja_En_Camino_E2, r1 := wire#w1)
   END_RUNG
   RUNG wire#powerrail
      Contact( #PhsMx )
      P_Trig( #MAUX_FP_En_camino_E2 )
   END_RUNG wire#w1
   // the same network as SCL:
   #_w1 := #PhsMx AND NOT #MAUX_FP_En_camino_E2;   // rising edge
   #MAUX_FP_En_camino_E2 := #PhsMx;
   IF #MAUX_PRV_Carga_OK_E2 THEN
       #MAUX_Caja_En_Camino_E2 := TRUE;   // SR flip-flop
   END_IF;
   IF #_w1 THEN #MAUX_Caja_En_Camino_E2 := FALSE; END_IF;
END_REGION

REGION Network 26: TIM Vaciado E1- Cuando no llega a la pHs
   RUNG wire#powerrail
      "FC911_CNT_Tiempo_UHS"(Temporizar := wire#w1, Valor_Tiempo := #V_Vaciado_E1, Base_tiempo_ms := 1, Valor_Actual := "DB230_CONTADORES".Mesa[#Mesa].CNT_AUSENCIA_ENTRADA, Tiempo_OK => #VaciadoE1_OK)
   END_RUNG
   RUNG wire#powerrail
      Contact( #MAUX_Caja_En_Camino_E1 )
      I_Contact( #PhsMx )
      Contact( "DB902_Estado_ZonaMesa".EstadoMesas[#Mesa].Marcha_CBx )
      I_Contact( "DB902_Estado_ZonaMesa".EstadoMesas[#Mesa].Error_CBx )
   END_RUNG wire#w1
   // the same network as SCL:
   "FC911_CNT_Tiempo_UHS"(Temporizar := #MAUX_Caja_En_Camino_E1 AND NOT #PhsMx AND "DB902_Estado_ZonaMesa".EstadoMesas[#Mesa].Marcha_CBx AND NOT "DB902_Estado_ZonaMesa".EstadoMesas[#Mesa].Error_CBx,
                          Valor_Tiempo := #V_Vaciado_E1,
                          Base_tiempo_ms := 1,
                          Valor_Actual := "DB230_CONTADORES".Mesa[#Mesa].CNT_AUSENCIA_ENTRADA,
                          Tiempo_OK => #VaciadoE1_OK);
END_REGION

REGION Network 27: TIM Vaciado E2- Cuando no llega a la pHs
   RUNG wire#powerrail
      "FC911_CNT_Tiempo_UHS"(Temporizar := wire#w1, Valor_Tiempo := #V_Vaciado_E2, Base_tiempo_ms := 1, Valor_Actual := "DB230_CONTADORES".Mesa[#Mesa].CNT_AUSENCIA_SALIDA, Tiempo_OK => #VaciadoE2_OK)
   END_RUNG
   RUNG wire#powerrail
      Contact( #MAUX_Caja_En_Camino_E2 )
      I_Contact( #PhsMx )
      Contact( "DB902_Estado_ZonaMesa".EstadoMesas[#Mesa].Marcha_CBx )
      I_Contact( "DB902_Estado_ZonaMesa".EstadoMesas[#Mesa].Error_CBx )
   END_RUNG wire#w1
   // the same network as SCL:
   "FC911_CNT_Tiempo_UHS"(Temporizar := #MAUX_Caja_En_Camino_E2 AND NOT #PhsMx AND "DB902_Estado_ZonaMesa".EstadoMesas[#Mesa].Marcha_CBx AND NOT "DB902_Estado_ZonaMesa".EstadoMesas[#Mesa].Error_CBx,
                          Valor_Tiempo := #V_Vaciado_E2,
                          Base_tiempo_ms := 1,
                          Valor_Actual := "DB230_CONTADORES".Mesa[#Mesa].CNT_AUSENCIA_SALIDA,
                          Tiempo_OK => #VaciadoE2_OK);
END_REGION

REGION Network 28: Si la caja enviada por E1 no llega despues de un tiempo, reseteamos
   RUNG wire#powerrail
      Contact( #VaciadoE1_OK )
      R_Coil( #MAUX_Caja_En_Camino_E1 )
   END_RUNG
   // the same network as SCL:
   IF #VaciadoE1_OK THEN #MAUX_Caja_En_Camino_E1 := FALSE; END_IF;
END_REGION

REGION Network 29: Si la caja enviada por E2 no llega despues de un tiempo, reseteamos
   RUNG wire#powerrail
      Contact( #VaciadoE2_OK )
      R_Coil( #MAUX_Caja_En_Camino_E2 )
   END_RUNG
   // the same network as SCL:
   IF #VaciadoE2_OK THEN #MAUX_Caja_En_Camino_E2 := FALSE; END_IF;
END_REGION
END_FUNCTION
